{attribute 'GeneratedUsingTerminal: EK1300-0000-0017'}
{attribute addProperty BoxType "EK1300-0000-0017"}
{attribute addProperty Id "UndervoltageAT %I*BOOL1"}
{attribute addProperty CRC "2984778146"}
{attribute addProperty Size "1"}
TYPE Status_Up_B1E819A2 EXTENDS InputBase_8311D824 :
STRUCT
	{attribute addProperty Name "Undervoltage"}
	Undervoltage AT %I* : BOOL;
END_STRUCT
END_TYPE

(* stored: Version 1.2.0.0, ProductVersion 3.1.4024.11
   DUT Status_Up_B1E819A2: Id {147ce706-7265-4db0-837c-c0bd1e016a00} *)
